(* CODESYS project LockChamber_student_valmis.project

Project tree, tasks and I/O mapping:
  Device : CODESYS Control Win V3, 3S - Smart Software Solutions GmbH, version 3.5.16.20
    application Application
      libraries: Standard, * (System); CmpVisuHandler, 3.5.16.10 (System)
      task MainTask (cyclic, interval t#10ms, priority 1) calls Model, POU
      task VISU_TASK (cyclic, interval 10 ms, priority 10) calls VisuElems.Visu_Prg
      program Model [ST]: gateMotionACT, levelControlACT, sensorsUpdateACT, initializationACT, blueBoatMoveACT, redBoatMoveACT
      image pool ImagePool
      visualisation Visualization
      global variables GVL
      program POU [SFC]: LevelDe_active, LeftGate_active, LeftIn_active, LeftGate2_active, LevelDe_exit, LevelIn_active, LevelIn_exit, RightGate_active, LeftOut_active, LevelDe_entry, LevelIn2_active, RightGate2_active, RightIn_active, RightGate3_active, LevelDe2_active, LeftGate3_active, LevelIn2_entry, LevelIn2_exit, LevelDe2_exit, Step8_active, Step8_active_0, ProcessRight_active, RightShip_entry, RightShip_exit, LeftShip_entry, LeftShip_exit, Wait_exit, Wait2_exit
  5ce3da45-db07-42e7-a21c-a00fff4ed8f6|C:\Users\Andrei\Desktop\ferry-157517_640.png
  text list GlobalTextList
  5ce3da45-db07-42e7-a21c-a00fff4ed8f6|C:\Users\Andrei\Desktop\ferry-157516_640.png
  5ce3da45-db07-42e7-a21c-a00fff4ed8f6|C:\Users\Andrei\Desktop\green arrow 2.png
  5ce3da45-db07-42e7-a21c-a00fff4ed8f6|C:\Users\Andrei\Desktop\green arrow.png
  5ce3da45-db07-42e7-a21c-a00fff4ed8f6|C:\Users\Andrei\Desktop\red arrow 2.png
  5ce3da45-db07-42e7-a21c-a00fff4ed8f6|C:\Users\Andrei\Desktop\red arrow.png
*)

// Device/Application/GVL
VAR_GLOBAL
	// Sensors:
	LeftClosed:BOOL;
	LeftOpen:BOOL;
	RightClosed:BOOL;
	RightOpen:BOOL;
	ShipFromLeft:BOOL;
	ShipFromRight:BOOL;
	ShipAtLeft:BOOL;
	ShipAtRight:BOOL;
	LowLevel:BOOL;
	HighLevel:BOOL;
	ShipInLock:BOOL;
	
	// Actuators:
	OpenLeft:BOOL;
	OpenRight:BOOL;
	IncreaseLevel:BOOL;
	DecreaseLevel:BOOL;
	FreeLeft:BOOL;
	FreeRight:BOOL;
END_VAR

// Device/Application/Model
PROGRAM Model
VAR
	// Change following variables as required.
	cycleTime :REAL := 10;
	gateSpeed :REAL := 50;
	fillingSpeed :REAL := 100;
	emptyingSpeed :REAL := 100;
	boatSpeed :REAL := 200;
END_VAR

VAR_INPUT
	// Input variables to the model.
	gateLeftOpen :BOOL;		// Open gate on the left.
	gateRightOpen :BOOL;	// Open gate on the right.
	increaseWater :BOOL;	// Open right valve.
	decreaseWater :BOOL;	// Open left valve.
	entryLeft :BOOL;		// Left semaphore.
	entryRight :BOOL;		// Right semaphore.
END_VAR
VAR_OUTPUT
	// Ouput variables from the model.
	gateLeftClosed :BOOL;
	gateRightClosed :BOOL;
	waterLow :BOOL;
	waterHigh :BOOL;
	shipFromLeft :BOOL;
	shipAtLeftGate :BOOL;
	shipInLock :BOOL;
	gateLeftOpened :BOOL;
	gateRightOpened :BOOL;
	shipAtRightGate :BOOL;
	shipFromRight :BOOL;
END_VAR

VAR
	// Model's internal variables. Do not change unless you know what you are doing.
	gatesInitialized :BOOL;
	gateLeftDown :ARRAY [0..3] OF VisuStructPoint;
	gateLeftUp :ARRAY [0..3] OF VisuStructPoint;
	gateLeftDownPos :ARRAY [0..3] OF REAL := [429,244,429,462];
	gateLeftUpPos :ARRAY [0..3] OF REAL := [429,462,429,244];
	gateRightDown :ARRAY [0..3] OF VisuStructPoint;
	gateRightUp :ARRAY [0..3] OF VisuStructPoint;
	gateRightDownPos :ARRAY [0..3] OF REAL := [790,244,790,462];
	gateRightUpPos :ARRAY [0..3] OF REAL := [790,462,790,244];
	waterLevel :REAL;
	
	boatRedPosX :REAL := -310;
	boatRedPosY :REAL := 0.0;
	boatRedRot :REAL;
	boatBluePosX :REAL := 280;
	boatBluePosY :REAL := 0.0;
	boatBlueRot :REAL;
	bothGatesOpen :BOOL;
	boatRedError :BOOL;
	boatBlueSemiError :BOOL;
	boatBlueError :BOOL;
	newFromLeft :BOOL :=TRUE;
	newFromRight :BOOL :=TRUE;
END_VAR

// Read inputs to the model.
gateLeftOpen := GVL.OpenLeft;
gateRightOpen := GVL.OpenRight;
increaseWater := GVL.IncreaseLevel;
decreaseWater := GVL.DecreaseLevel;
entryLeft := GVL.FreeLeft;
entryRight := GVL.FreeRight;


// Initialization. Done once.
IF NOT(gatesInitialized) THEN
	initializationACT();
	gatesInitialized := TRUE;
END_IF

// Gate control
gateMotionACT();

// Water level control
levelControlACT();

// Red boat movement
redBoatMoveACT();

// Blue boat moevement
blueBoatMoveACT();

// Update status of sensors
sensorsUpdateACT();

// Output information from model.
GVL.LeftClosed := gateLeftClosed;
GVL.LeftOpen := gateLeftOpened;
GVL.RightClosed := gateRightClosed;
GVL.RightOpen := gateRightOpened;
GVL.ShipFromLeft := shipFromLeft;
GVL.ShipFromRight := shipFromRight;
GVL.ShipAtLeft := shipAtLeftGate;
GVL.ShipAtRight := shipAtRightGate;
GVL.LowLevel := waterLow;
GVL.HighLevel := waterHigh;
GVL.ShipInLock := shipInLock;

ACTION gateMotionACT:
// Open left gate motion.
IF gateLeftOpen THEN
	IF gateLeftDownPos[1] < gateLeftDown[3].iY THEN
		// Upper point of bottom gate.
		gateLeftDownPos[1] := gateLeftDownPos[1] + gateSpeed * cycleTime / 1000;
		gateLeftDown[0].iY := REAL_TO_INT(gateLeftDownPos[1]);
		gateLeftDownPos[0] := gateLeftDownPos[0] - 3 * gateSpeed * cycleTime / 1000;
		gateLeftDown[0].iX := REAL_TO_INT(gateLeftDownPos[0]);
		// Lower point of botom gate.
		gateLeftDownPos[3] := gateLeftDownPos[3] + 1.7857 * gateSpeed * cycleTime / 1000;
		gateLeftDown[1].iY := REAL_TO_INT(gateLeftDownPos[3]);
		gateLeftDownPos[2] := gateLeftDownPos[2] - 3 * gateSpeed * cycleTime / 1000;
		gateLeftDown[1].iX := REAL_TO_INT(gateLeftDownPos[2]);
	END_IF
	
	IF gateLeftUpPos[3] > gateLeftUp[0].iY THEN
		// Upper point of upper gate.
		gateLeftUpPos[3] := gateLeftUpPos[3] - gateSpeed * cycleTime / 1000;
		gateLeftUp[3].iY := REAL_TO_INT(gateLeftUpPos[3]);
		gateLeftUpPos[2] := gateLeftUpPos[2] - 1 * gateSpeed * cycleTime / 1000;
		gateLeftUp[3].iX := REAL_TO_INT(gateLeftUpPos[2]);
		// Lower point of upper gate.
		gateLeftUpPos[1] := gateLeftUpPos[1] - 2.04 * gateSpeed * cycleTime / 1000;
		gateLeftUp[2].iY := REAL_TO_INT(gateLeftUpPos[1]);
		gateLeftUpPos[0] := gateLeftUpPos[0] - 1 * gateSpeed * cycleTime / 1000;
		gateLeftUp[2].iX := REAL_TO_INT(gateLeftUpPos[0]);
	END_IF
ELSE
	IF gateLeftDownPos[1] > 244 THEN
		// Upper point of bottom gate.
		gateLeftDownPos[1] := gateLeftDownPos[1] - gateSpeed * cycleTime / 1000;
		gateLeftDown[0].iY := REAL_TO_INT(gateLeftDownPos[1]);
		gateLeftDownPos[0] := gateLeftDownPos[0] + 3 * gateSpeed * cycleTime / 1000;
		gateLeftDown[0].iX := REAL_TO_INT(gateLeftDownPos[0]);
		// Lower point of botom gate.
		gateLeftDownPos[3] := gateLeftDownPos[3] - 1.7857 * gateSpeed * cycleTime / 1000;
		gateLeftDown[1].iY := REAL_TO_INT(gateLeftDownPos[3]);
		gateLeftDownPos[2] := gateLeftDownPos[2] + 3 * gateSpeed * cycleTime / 1000;
		gateLeftDown[1].iX := REAL_TO_INT(gateLeftDownPos[2]);
	END_IF
	
	IF gateLeftUpPos[3] < 244 THEN
		// Upper point of upper gate.
		gateLeftUpPos[3] := gateLeftUpPos[3] + gateSpeed * cycleTime / 1000;
		gateLeftUp[3].iY := REAL_TO_INT(gateLeftUpPos[3]);
		gateLeftUpPos[2] := gateLeftUpPos[2] + 1 * gateSpeed * cycleTime / 1000;
		gateLeftUp[3].iX := REAL_TO_INT(gateLeftUpPos[2]);
		// Lower point of upper gate.
		gateLeftUpPos[1] := gateLeftUpPos[1] + 2.04 * gateSpeed * cycleTime / 1000;
		gateLeftUp[2].iY := REAL_TO_INT(gateLeftUpPos[1]);
		gateLeftUpPos[0] := gateLeftUpPos[0] + 1 * gateSpeed * cycleTime / 1000;
		gateLeftUp[2].iX := REAL_TO_INT(gateLeftUpPos[0]);
	END_IF
END_IF

// Open right gate motion
IF gateRightOpen THEN
	IF gateRightDownPos[1] < gateRightDown[3].iY THEN
		// Upper point of bottom gate
		gateRightDownPos[1] := gateRightDownPos[1] + gateSpeed * cycleTime / 1000;
		gateRightDown[0].iY := REAL_TO_INT(gateRightDownPos[1]);
		gateRightDownPos[0] := gateRightDownPos[0] - 1.5 * gateSpeed * cycleTime / 1000;
		gateRightDown[0].iX := REAL_TO_INT(gateRightDownPos[0]);
		// Lower point of bottom gate
		gateRightDownPos[3] := gateRightDownPos[3] + 1.7857 * gateSpeed * cycleTime / 1000;
		gateRightDown[1].iY := REAL_TO_INT(gateRightDownPos[3]);
		gateRightDownPos[2] := gateRightDownPos[2] - 1.5 * gateSpeed * cycleTime / 1000;
		gateRightDown[1].iX := REAL_TO_INT(gateRightDownPos[2]);
	END_IF
	
	IF gateRightUpPos[3] > gateRightUp[0].iY THEN
		// Upper point of top gate
		gateRightUpPos[3] := gateRightUpPos[3] - gateSpeed * cycleTime / 1000;
		gateRightUp[3].iY := REAL_TO_INT(gateRightUpPos[3]);
		gateRightUpPos[2] := gateRightUpPos[2] - 2.3 * gateSpeed * cycleTime / 1000;
		gateRightUp[3].iX := REAL_TO_INT(gateRightUpPos[2]);
		// Lower point of top gate
		gateRightUpPos[1] := gateRightUpPos[1] - 2.04 * gateSpeed * cycleTime / 1000;
		gateRightUp[2].iY := REAL_TO_INT(gateRightUpPos[1]);
		gateRightUpPos[0] := gateRightUpPos[0] - 2.3 * gateSpeed * cycleTime / 1000;
		gateRightUp[2].iX := REAL_TO_INT(gateRightUpPos[0]);
	END_IF
ELSE
	IF gateRightDownPos[1] > 244 THEN
		// Upper point of bottom gate
		gateRightDownPos[1] := gateRightDownPos[1] - gateSpeed * cycleTime / 1000;
		gateRightDown[0].iY := REAL_TO_INT(gateRightDownPos[1]);
		gateRightDownPos[0] := gateRightDownPos[0] + 1.5 * gateSpeed * cycleTime / 1000;
		gateRightDown[0].iX := REAL_TO_INT(gateRightDownPos[0]);
		// Lower point of bottom gate
		gateRightDownPos[3] := gateRightDownPos[3] - 1.7857 * gateSpeed * cycleTime / 1000;
		gateRightDown[1].iY := REAL_TO_INT(gateRightDownPos[3]);
		gateRightDownPos[2] := gateRightDownPos[2] + 1.5 * gateSpeed * cycleTime / 1000;
		gateRightDown[1].iX := REAL_TO_INT(gateRightDownPos[2]);
	END_IF
	
	IF gateRightUpPos[3] < 244 THEN
		// Upper point of top gate
		gateRightUpPos[3] := gateRightUpPos[3] + gateSpeed * cycleTime / 1000;
		gateRightUp[3].iY := REAL_TO_INT(gateRightUpPos[3]);
		gateRightUpPos[2] := gateRightUpPos[2] + 2.3 * gateSpeed * cycleTime / 1000;
		gateRightUp[3].iX := REAL_TO_INT(gateRightUpPos[2]);
		// Lower point of top gate
		gateRightUpPos[1] := gateRightUpPos[1] + 2.04 * gateSpeed * cycleTime / 1000;
		gateRightUp[2].iY := REAL_TO_INT(gateRightUpPos[1]);
		gateRightUpPos[0] := gateRightUpPos[0] + 2.3 * gateSpeed * cycleTime / 1000;
		gateRightUp[2].iX := REAL_TO_INT(gateRightUpPos[0]);
	END_IF
END_IF
END_ACTION

ACTION levelControlACT:
// Function to increase or decrease the level in the lock chamber
// Increase level with valve.
IF increaseWater AND NOT(decreaseWater) AND waterLevel > -131.0 AND gateLeftClosed THEN
	waterLevel := waterLevel - fillingSpeed * cycleTime / 1000;
END_IF

// Decrease level with valve.
IF decreaseWater AND NOT(increaseWater) AND waterLevel < 0.1 AND gateRightClosed THEN
	waterLevel := waterLevel + emptyingSpeed * cycleTime / 1000;
END_IF

// If left gate is not closed and right gate is closed, decrease water level fast.
IF NOT(gateLeftClosed) AND gateRightClosed THEN
	IF waterLevel + 1.5 < 0 THEN
		waterLevel := waterLevel + 1.5;
	ELSE
		waterLevel := 0.0;
	END_IF
END_IF

// If left gate is closed and right gate is open, increase the water level fast.
IF gateLeftClosed AND NOT(gateRightClosed) THEN
	IF waterLevel - 1.5 > -131 THEN
		waterLevel := waterLevel - 1.5;
	ELSE
		waterLevel := -131;
	END_IF
END_IF

// If both gates are not completly closed, water "flows from one level to another".
IF NOT(gateLeftClosed) AND NOT(gateRightClosed) THEN
	bothGatesOpen := TRUE;
	waterLevel := 0.0;
END_IF
IF gateLeftClosed OR gateRightClosed THEN
	bothGatesOpen := FALSE;
END_IF
END_ACTION

ACTION sensorsUpdateACT:
// Function used to update status of sensors.
// Gate on the left is closed.
IF gateLeftDownPos[0] > 428.9 THEN
	gateLeftClosed := TRUE;
ELSE
	gateLeftClosed := FALSE;
END_IF

// Gate on the right is closed.
IF gateRightDownPos[0] > 789.9 THEN
	gateRightClosed := TRUE;
ELSE
	gateRightClosed := FALSE;
END_IF

// Water level high.
IF waterLevel < -130.9 THEN
	waterHigh := TRUE;
ELSE
	waterHigh := FALSE;
END_IF

// Water level low.
IF waterLevel > -0.1 THEN
	waterLow := TRUE;
ELSE
	waterLow := FALSE;
END_IF

// Ship from left.
IF boatRedPosX > 29 AND boatRedPosX < 440 THEN
	shipFromLeft := TRUE;
ELSE
	shipFromLeft := FALSE;
END_IF

// Ship at the left gate.
IF (boatRedPosX > 140 AND boatRedPosX < 425) OR (boatBluePosX < -480
 AND boatBluePosX > -760) THEN
	shipAtLeftGate := TRUE;
ELSE
	shipAtLeftGate := FALSE;
END_IF

// Ship in the lock-gate.
IF (boatRedPosX > 464 AND boatRedPosX < 790) OR (boatBluePosX < -454
 AND boatBluePosX > -780) THEN
	shipInLock := TRUE;
ELSE
	shipInLock := FALSE;
END_IF

// Gate on the left is opened.
IF gateLeftDownPos[0] < 345.1 THEN
	gateLeftOpened := TRUE;
ELSE
	gateLeftOpened := FALSE;
END_IF

// Gate on the right is opened.
IF gateRightDownPos[0] < 748.1 THEN
	gateRightOpened := TRUE;
ELSE
	gateRightOpened := FALSE;
END_IF

// Ship at the right gate.
IF (boatRedPosX > 510 AND boatRedPosX < 790) OR (boatBluePosX < -135
 AND boatBluePosX > -415) THEN
	shipAtRightGate := TRUE;
ELSE
	shipAtRightGate := FALSE;
END_IF

// Ship from right.
IF boatBluePosX < -29 AND boatBluePosX > -420 THEN
	shipFromRight := TRUE;
ELSE
	shipFromRight := FALSE;
END_IF
END_ACTION

ACTION initializationACT:
// Initialize points with original coordinates.
// Left gates points.
	gateLeftDown[0].iX := 429;
	gateLeftDown[0].iY := 244;
	gateLeftDown[1].iX := 429;
	gateLeftDown[1].iY := 462;
	gateLeftDown[2].iX := 410;
	gateLeftDown[2].iY := 512;
	gateLeftDown[3].iX := 410;
	gateLeftDown[3].iY := 272;
	gateLeftUp[0].iX := 445;
	gateLeftUp[0].iY := 219;
	gateLeftUp[1].iX := 445;
	gateLeftUp[1].iY := 411;
	gateLeftUp[2].iX := 429;
	gateLeftUp[2].iY := 462;
	gateLeftUp[3].iX := 429;
	gateLeftUp[3].iY := 244;
	
// Right gates points.
	gateRightDown[0].iX := 790;
	gateRightDown[0].iY := 244;
	gateRightDown[1].iX := 790;
	gateRightDown[1].iY := 462;
	gateRightDown[2].iX := 810;
	gateRightDown[2].iY := 512;
	gateRightDown[3].iX := 810;
	gateRightDown[3].iY := 272;
	gateRightUp[0].iX := 775;
	gateRightUp[0].iY := 219;
	gateRightUp[1].iX := 775;
	gateRightUp[1].iY := 411;
	gateRightUp[2].iX := 790;
	gateRightUp[2].iY := 462;
	gateRightUp[3].iX := 790;
	gateRightUp[3].iY := 244;
END_ACTION

ACTION blueBoatMoveACT:
// Boat enters the scene from the right.
IF boatBluePosX > -30 THEN
	boatBluePosX := boatBluePosX - boatSpeed * cycleTime / 1000;
END_IF

// While right green light is on and right gate is opened,
// boat goes inside the lock chamber.
IF entryRight AND gateRightOpened AND boatBluePosX > -455 AND boatBluePosX < -29
 AND NOT(boatBlueError) THEN
	boatBluePosX := boatBluePosX - boatSpeed * cycleTime / 1000;
END_IF

// Exit the lock chamber once the water low level is reached and
// left gates are open and continue going once out of the chamber.
IF (boatBluePosX < -420 AND waterLow AND gateLeftOpened AND NOT(boatBlueError)
 OR (boatBluePosX < -780)) AND boatBluePosX > -1205 THEN
	boatBluePosX := boatBluePosX - boatSpeed * cycleTime / 1000;
END_IF

// Once boat exists the scene from the right, return it to origin.
IF boatBluePosX < -1200 and newFromRight THEN
	boatBluePosY := 0.0;
	boatBluePosX := 280;
END_IF

// This part takes care of the error state when both gates are open.
IF boatBluePosX < -240 AND boatBluePosX > -641 AND (bothGatesOpen OR boatBlueError) THEN
	boatBlueError := TRUE;
	boatBlueRot := -15;
	boatBluePosX := boatBluePosX - 1;
	boatBluePosY := boatBluePosY + 0.5;
END_IF
IF boatBluePosX < -640 AND boatBlueError THEN
	IF boatBluePosY < 190 THEN
		boatBluePosX := boatBluePosX - 0.1;
		boatBluePosY := boatBluePosY + 0.3;
		boatBlueRot := - 10 * SIN(boatBluePosY / 10);
	END_IF
END_IF

// While inside the lock chamber, boat moves with water level.
// should be under the rest of functions here in order to get the error in time.
IF boatBluePosX < -270 AND BoatBluePosX > -625 AND NOT(boatBlueError) AND NOT(boatBlueSemiError) THEN
	boatBluePosY := 131 + waterLevel;
END_IF
END_ACTION

ACTION redBoatMoveACT:
// Boat enters the scene.
IF boatRedPosX < 30 AND NOT(boatRedError) THEN
	boatRedPosX := boatRedPosX + boatSpeed * cycleTime / 1000;
END_IF

// While left green light is on and left gate is open, boat goes into the lock chamber.
IF entryLeft AND gateLeftOpened AND boatRedPosX > 29 AND boatRedPosX < 465
 AND NOT(boatRedError) THEN
	boatRedPosX := boatRedPosX + boatSpeed * cycleTime / 1000;
END_IF

// While inside the lock chamber, boat moves with the water level.
IF boatRedPosX > 310 AND boatRedPosX < 515  AND NOT(boatRedError) THEN
	boatRedPosY := waterLevel;
END_IF

// Exit from lock chamber once water high level is reached and right gates
// are opened.
IF ((boatRedPosX > 425 AND waterHigh AND gateRightOpened  AND NOT(boatRedError))
 OR (boatRedPosX > 770)) AND (boatRedPosX < 1205) THEN
	boatRedPosX := boatRedPosX + boatSpeed * cycleTime / 1000;
END_IF

// Once boat exists the scene from the right, return it to origin.
IF boatRedPosX > 1200 AND newFromLeft THEN
	boatRedPosY := 0.0;
	boatRedPosX := -310.0;
END_IF

// This part takes care of the error state when both gates are open.
IF boatRedPosX > 260 AND boatRedPosX < 690 AND bothGatesOpen OR boatRedError THEN
	boatRedError := TRUE;
	IF boatRedPosY < 65 THEN
		boatRedRot := 10 * SIN(boatRedPosY/10);
		boatRedPosX := boatRedPosX + 0.1;
		boatRedPosY := boatRedPosY + 0.3;
	END_IF
END_IF
END_ACTION

END_PROGRAM

// Device/Application/POU
PROGRAM POU
VAR
	process:BOOL := FALSE;
	
END_VAR

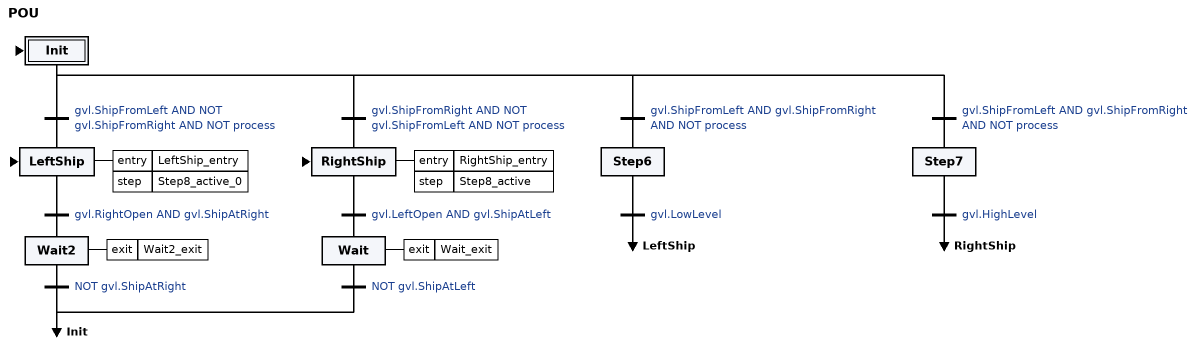
INITIAL_STEP Init:
END_STEP
TRANSITION FROM Init TO LeftShip
    := gvl.ShipFromLeft AND NOT gvl.ShipFromRight AND NOT process;
END_TRANSITION
STEP LeftShip:
    LeftShip_entry(P1);  // entry action
    Step8_active_0(N);  // step action
END_STEP
TRANSITION FROM LeftShip TO Wait2
    := gvl.RightOpen AND gvl.ShipAtRight;
END_TRANSITION
STEP Wait2:
    Wait2_exit(P0);  // exit action
END_STEP
TRANSITION FROM Wait2 TO Init
    := NOT gvl.ShipAtRight;
END_TRANSITION
TRANSITION FROM Init TO RightShip
    := gvl.ShipFromRight AND NOT gvl.ShipFromLeft AND NOT process;
END_TRANSITION
STEP RightShip:
    RightShip_entry(P1);  // entry action
    Step8_active(N);  // step action
END_STEP
TRANSITION FROM RightShip TO Wait
    := gvl.LeftOpen AND gvl.ShipAtLeft;
END_TRANSITION
STEP Wait:
    Wait_exit(P0);  // exit action
END_STEP
TRANSITION FROM Wait TO Init
    := NOT gvl.ShipAtLeft;
END_TRANSITION
TRANSITION FROM Init TO Step6
    := gvl.ShipFromLeft AND gvl.ShipFromRight AND NOT process;
END_TRANSITION
TRANSITION FROM Init TO Step7
    := gvl.ShipFromLeft AND gvl.ShipFromRight AND NOT process;
END_TRANSITION
STEP Step7:
END_STEP
TRANSITION FROM Step7 TO RightShip
    := gvl.HighLevel;
END_TRANSITION
STEP Step6:
END_STEP
TRANSITION FROM Step6 TO LeftShip
    := gvl.LowLevel;
END_TRANSITION

ACTION LevelDe_active:
gvl.DecreaseLevel := TRUE;
END_ACTION

ACTION LeftGate_active:
gvl.OpenLeft := TRUE;
END_ACTION

ACTION LeftIn_active:
gvl.FreeLeft := TRUE;
END_ACTION

ACTION LeftGate2_active:
gvl.OpenLeft := FALSE;
END_ACTION

ACTION LevelDe_exit:
gvl.DecreaseLevel := FALSE;
END_ACTION

ACTION LevelIn_active:
gvl.IncreaseLevel := TRUE;
END_ACTION

ACTION LevelIn_exit:
gvl.IncreaseLevel := FALSE;
END_ACTION

ACTION RightGate_active:
gvl.OpenRight := TRUE;
END_ACTION

ACTION LeftOut_active:

END_ACTION

ACTION LevelDe_entry:
gvl.OpenRight := FALSE;
END_ACTION

ACTION LevelIn2_active:
gvl.IncreaseLevel := TRUE;
END_ACTION

ACTION RightGate2_active:
gvl.OpenRight := TRUE;
END_ACTION

ACTION RightIn_active:
gvl.FreeRight := TRUE;
END_ACTION

ACTION RightGate3_active:
gvl.OpenRight := FALSE;
END_ACTION

ACTION LevelDe2_active:
gvl.DecreaseLevel := TRUE;
END_ACTION

ACTION LeftGate3_active:
gvl.OpenLeft := TRUE;
END_ACTION

ACTION LevelIn2_entry:
gvl.OpenLeft := FALSE;
END_ACTION

ACTION LevelIn2_exit:
gvl.IncreaseLevel := FALSE;
END_ACTION

ACTION LevelDe2_exit:
gvl.DecreaseLevel := FALSE;
END_ACTION

ACTION Step8_active:
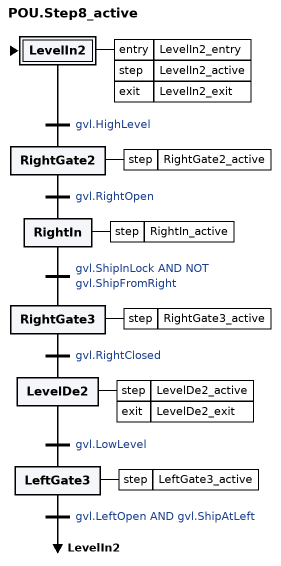
INITIAL_STEP LevelIn2:
    LevelIn2_entry(P1);  // entry action
    LevelIn2_active(N);  // step action
    LevelIn2_exit(P0);  // exit action
END_STEP
TRANSITION FROM LevelIn2 TO RightGate2
    := gvl.HighLevel;
END_TRANSITION
STEP RightGate2:
    RightGate2_active(N);  // step action
END_STEP
TRANSITION FROM RightGate2 TO RightIn
    := gvl.RightOpen;
END_TRANSITION
STEP RightIn:
    RightIn_active(N);  // step action
END_STEP
TRANSITION FROM RightIn TO RightGate3
    := gvl.ShipInLock AND NOT gvl.ShipFromRight;
END_TRANSITION
STEP RightGate3:
    RightGate3_active(N);  // step action
END_STEP
TRANSITION FROM RightGate3 TO LevelDe2
    := gvl.RightClosed;
END_TRANSITION
STEP LevelDe2:
    LevelDe2_active(N);  // step action
    LevelDe2_exit(P0);  // exit action
END_STEP
TRANSITION FROM LevelDe2 TO LeftGate3
    := gvl.LowLevel;
END_TRANSITION
STEP LeftGate3:
    LeftGate3_active(N);  // step action
END_STEP
TRANSITION FROM LeftGate3 TO LevelIn2
    := gvl.LeftOpen AND gvl.ShipAtLeft;
END_TRANSITION
END_ACTION

ACTION Step8_active_0:
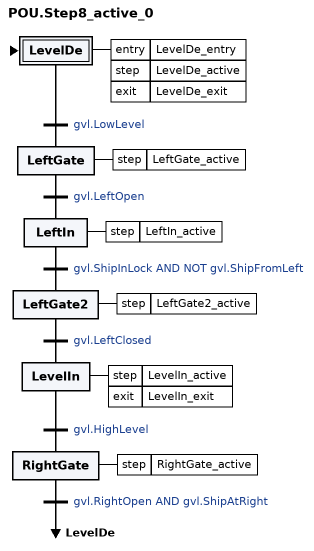
INITIAL_STEP LevelDe:
    LevelDe_entry(P1);  // entry action
    LevelDe_active(N);  // step action
    LevelDe_exit(P0);  // exit action
END_STEP
TRANSITION FROM LevelDe TO LeftGate
    := gvl.LowLevel;
END_TRANSITION
STEP LeftGate:
    LeftGate_active(N);  // step action
END_STEP
TRANSITION FROM LeftGate TO LeftIn
    := gvl.LeftOpen;
END_TRANSITION
STEP LeftIn:
    LeftIn_active(N);  // step action
END_STEP
TRANSITION FROM LeftIn TO LeftGate2
    := gvl.ShipInLock AND NOT gvl.ShipFromLeft;
END_TRANSITION
STEP LeftGate2:
    LeftGate2_active(N);  // step action
END_STEP
TRANSITION FROM LeftGate2 TO LevelIn
    := gvl.LeftClosed;
END_TRANSITION
STEP LevelIn:
    LevelIn_active(N);  // step action
    LevelIn_exit(P0);  // exit action
END_STEP
TRANSITION FROM LevelIn TO RightGate
    := gvl.HighLevel;
END_TRANSITION
STEP RightGate:
    RightGate_active(N);  // step action
END_STEP
TRANSITION FROM RightGate TO LevelDe
    := gvl.RightOpen AND gvl.ShipAtRight;
END_TRANSITION
END_ACTION

ACTION ProcessRight_active:
process := TRUE;
END_ACTION

ACTION RightShip_entry:
process := TRUE;
END_ACTION

ACTION RightShip_exit:
process := FALSE;
END_ACTION

ACTION LeftShip_entry:
process := TRUE;
END_ACTION

ACTION LeftShip_exit:
process := FALSE;
END_ACTION

ACTION Wait_exit:
process := FALSE;
END_ACTION

ACTION Wait2_exit:
process := FALSE;
END_ACTION

END_PROGRAM

// Device/Application/Visualization
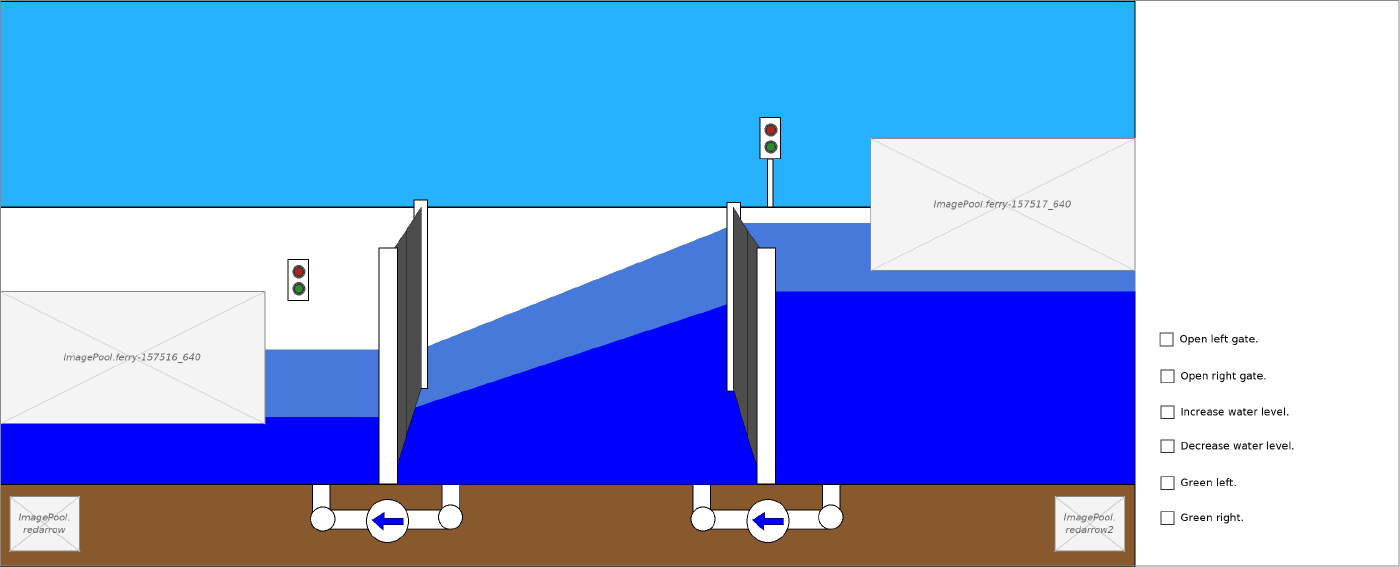
VISUALIZATION Visualization  // 1480x600
    Rectangle (0,1 1200x218)
    Rectangle (0,512 1200x88)
    Rectangle (0,410 1200x102)
    Rectangle (0,219 1200x190)
    Polygon (773,236) (781,408) (813,512) (1200,512) (1200,236)
    Polygon (774,236) (808,308) (1200,308) (1200,236)
    Rectangle (742,539 136x21)
    Rectangle (869,512 19x26)
    Ellipse (865,534 26x26)
    Rectangle (732,512 19x33)
    Ellipse (730,536 26x26)
    Ellipse (789,528 45x46)
    Polygon (808,542) (795,550) (807,561) (807,555) (828,555) (828,548) (808,548), invisible if: NOT(Model.increaseWater)
    Rectangle (340,539 136x21)
    Rectangle (467,512 19x26)
    Ellipse (463,534 26x26)
    Rectangle (330,512 19x33)
    Ellipse (328,536 26x26)
    Ellipse (387,528 45x46)
    Polygon (406,542) (393,550) (405,561) (405,555) (426,555) (426,548) (406,548), invisible if: NOT(Model.decreaseWater)
    RoundedRectangle (803,124 22x44)
    Lamp1 (807,129 16x17), variable: NOT(Model.entryRight), style: Lamp-Lamp1-Red
    Rectangle (811,168 6x51)
    Lamp1 (807,147 16x17), variable: Model.entryRight, style: Lamp-Lamp1-Green
    RoundedRectangle (304,274 22x44)
    Lamp1 (308,279 16x17), variable: NOT(Model.entryLeft), style: Lamp-Lamp1-Red
    Lamp1 (308,297 16x17), variable: Model.entryLeft, style: Lamp-Lamp1-Green
    Checkbox (1224,344 273x30), "Open left gate.", variable: GVL.OpenLeft
    Checkbox (1225,383 273x30), "Open right gate.", variable: GVL.OpenRight
    Checkbox (1225,421 273x30), "Increase water level.", variable: GVL.IncreaseLevel
    Checkbox (1225,457 273x30), "Decrease water level.", variable: GVL.DecreaseLevel
    Checkbox (1225,496 273x30), "Green left.", variable: GVL.FreeLeft
    Checkbox (1225,533 273x30), "Green right.", variable: GVL.FreeRight
    Polygon (0,512) (0,437) (1,370) (444,370) (443,410) (409,512)
    Polygon (445,370) (409,441) (0,441) (0,370)
    Polygon (445,369) (410,440) (809,440) (775,369), invisible if: Model.bothGatesOpen
        p2738717112: Model.waterLevel
    Polygon (445,369) (410,440) (809,309) (775,238), invisible if: NOT(Model.bothGatesOpen)
        p2738717112: Model.waterLevel
    Polygon (408,441) (811,308) (811,512) (408,512), invisible if: NOT(Model.bothGatesOpen)
    Rectangle (408,440 403x72), invisible if: Model.bothGatesOpen
        p2773130477: Model.waterLevel
    RoundedRectangle (768,214 15x200)
    RoundedRectangle (437,211 15x200)
    Polygon (445,219) (445,411) (429,462) (429,244)
        p1285906596: ADR(Model.gateLeftUp)
    Polygon (775,219) (775,411) (790,462) (790,244)
        p1285906596: ADR(Model.gateRightUp)
    Image (920,146 280x140), image: ImagePool.ferry-157517_640
        p3560616238: Model.boatBluePosX
        p2738717112: Model.boatBluePosY
        p2858320360: Model.boatBlueRot
    Image (0,308 280x140), image: ImagePool.ferry-157516_640
        p3560616238: Model.boatRedPosX
        p2738717112: Model.boatRedPosY
        p2858320360: Model.boatRedRot
    Polygon (429,244) (429,462) (414,513) (410,272)
        p1285906596: ADR(Model.gateLeftDown)
    Polygon (790,244) (790,462) (806,513) (810,272)
        p1285906596: ADR(Model.gateRightDown)
    RoundedRectangle (400,262 20x250)
    RoundedRectangle (800,262 20x250)
    Rectangle (1201,137 279x173)
    Image (10,525 74x58), image: ImagePool.greenarrow
        OnMouseDown: execute { Model.newFromLeft := FALSE; }
    Image (10,525 74x58), invisible if: Model.newFromLeft, image: ImagePool.redarrow
        OnMouseDown: execute { Model.newFromLeft := TRUE; }
    Image (1115,525 74x58), image: ImagePool.greenarrow2
        OnMouseDown: execute { Model.newFromRight := FALSE; }
    Image (1115,525 74x58), invisible if: Model.newFromRight, image: ImagePool.redarrow2
        OnMouseDown: execute { Model.newFromRight := TRUE; }
END_VISUALIZATION
